ABB RobotStudio station: Sesion7_Parte1_interrupciones.rspag

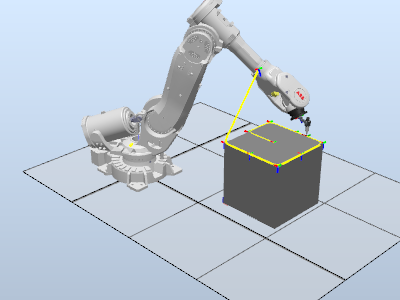
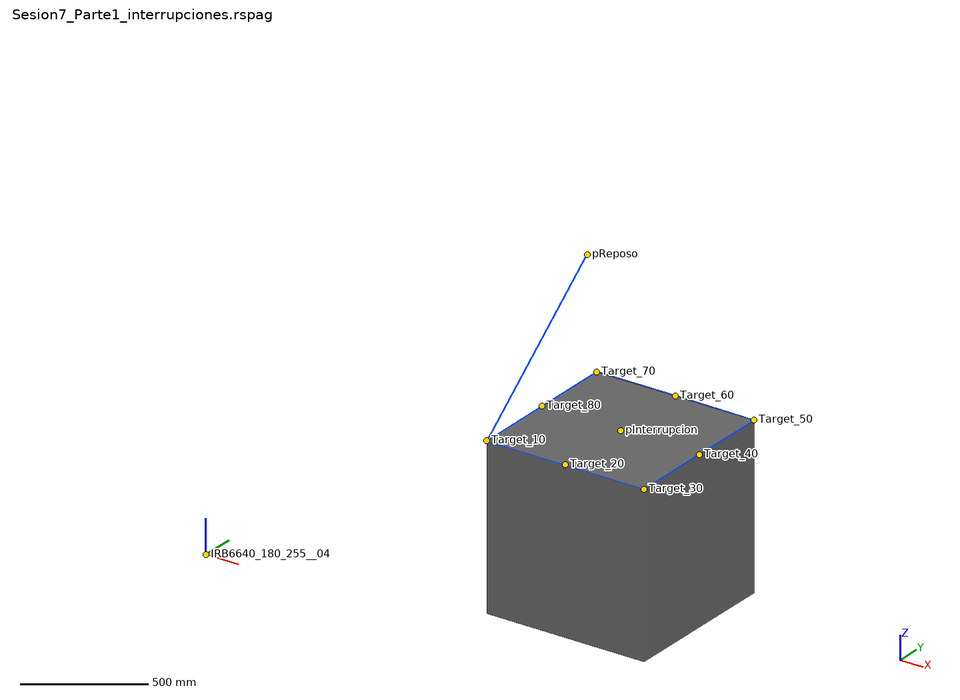
[picture v1: parts stored in the station drawn from their meshes, with robot base, taught points and paths (robot models come from the ABB library and are not in the file)]
--- station ---
Station borr (saved by RobotStudio 24.1.10713.1)
Controller Controlador10
  mechanical unit ROB_1: IRB6640_180_255__04, 6 joints, base frame (0, 0, 0) mm
Layout (positions relative to the parent item):
  - IRB6640_180_255__04 [mechanism, from %ABB.RobotStudio.Models.IRB6640%\IRB6640_180_255_G_04.rslib] at (0, 0, 0) mm; joint values [0.569, 0.4564, 0.2981, -0.9875, 0.4087, 1.4142] (rad or m)
  - MyTool [mechanism, from Training Objects\myTool.rslib] at (1608.5, 950, 950.53) mm, rotated rx -180 ry 38 rz 180 deg
  - Pieza_1 [part], size 750 x 750 x 750 mm
Attachment: MyTool is attached to IRB6640_180_255__04 / Link6
Targets, tools, work objects and paths stored in the station and not in the controller backup, written as RAPID:
! task T_ROB1
MODULE Module1
  PROC Path_10()
    MoveL pReposo,v1000,z100,MyTool\WObj:=wobj0;
    MoveL Target_10,v1000,z100,MyTool\WObj:=Workobject_1;
    MoveL Target_20,v1000,z100,MyTool\WObj:=Workobject_1;
    MoveL Target_30,v1000,z100,MyTool\WObj:=Workobject_1;
    MoveL Target_40,v1000,z100,MyTool\WObj:=Workobject_1;
    MoveL Target_50,v1000,z100,MyTool\WObj:=Workobject_1;
    MoveL Target_60,v1000,z100,MyTool\WObj:=Workobject_1;
    MoveL Target_70,v1000,z100,MyTool\WObj:=Workobject_1;
    MoveL Target_80,v1000,z100,MyTool\WObj:=Workobject_1;
    MoveL pInterrupcion,v1000,z100,MyTool\WObj:=Workobject_1;
  ENDPROC
ENDMODULE


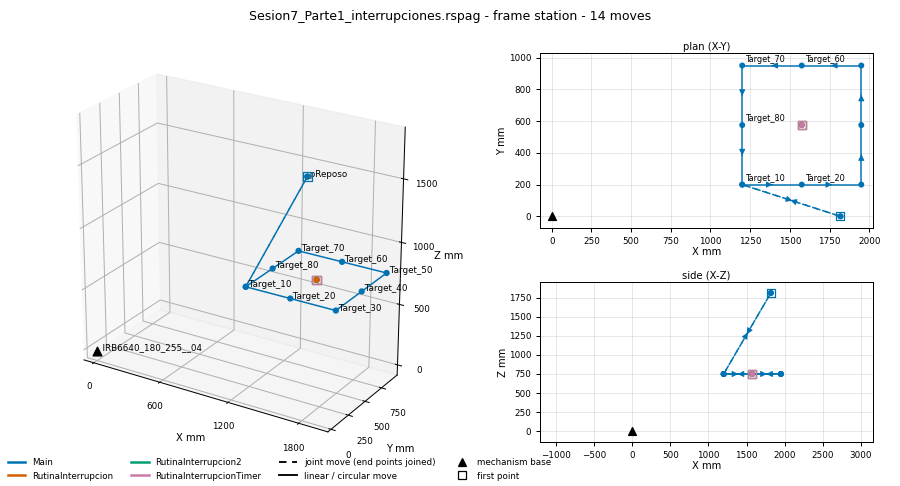
[picture p0: tool path of Sesion7_Parte1_interrupciones.rspag in frame station, 14 of 17 moves have a stored position in this frame; points joined in program order, loops and branches not executed]
--- Backups/Controlador10/RAPID/TASK1/PROGMOD/CalibData.mod ---
MODULE CalibData
    PERS tooldata MyTool:=[TRUE,[[31.792631019,0,229.638935148],[0.945518576,0,0.325568154,0]],[1,[0,0,1],[1,0,0,0],0,0,0]];
    TASK PERS wobjdata Workobject_1:=[FALSE,TRUE,"",[[1200,200,0],[1,0,0,0]],[[0,0,0],[1,0,0,0]]];
ENDMODULE

--- Backups/Controlador10/RAPID/TASK1/PROGMOD/Module1.mod ---
MODULE Module1
    CONST robtarget pReposo:=[[1818.681916784,0,1812.64730631],[0.190808996,0,0.981627183,0],[0,0,0,0],[9E+09,9E+09,9E+09,9E+09,9E+09,9E+09]];
    CONST robtarget Target_10:=[[0,0,750],[0,0,1,0],[0,-1,0,0],[9E+09,9E+09,9E+09,9E+09,9E+09,9E+09]];
    CONST robtarget Target_20:=[[375,0,750],[0,0,1,0],[0,-1,0,0],[9E+09,9E+09,9E+09,9E+09,9E+09,9E+09]];
    CONST robtarget Target_30:=[[750,0,750],[0,0,1,0],[0,-1,0,0],[9E+09,9E+09,9E+09,9E+09,9E+09,9E+09]];
    CONST robtarget Target_40:=[[750,375,750],[0,0,1,0],[0,-1,0,0],[9E+09,9E+09,9E+09,9E+09,9E+09,9E+09]];
    CONST robtarget Target_50:=[[750,750,750],[0,0,1,0],[0,-1,0,0],[9E+09,9E+09,9E+09,9E+09,9E+09,9E+09]];
    CONST robtarget Target_60:=[[375,750,750],[0,0,1,0],[0,-1,0,0],[9E+09,9E+09,9E+09,9E+09,9E+09,9E+09]];
    CONST robtarget Target_70:=[[0,750,750],[0,0,1,0],[0,0,0,0],[9E+09,9E+09,9E+09,9E+09,9E+09,9E+09]];
    CONST robtarget Target_80:=[[0,375,750],[0,0,1,0],[0,0,0,0],[9E+09,9E+09,9E+09,9E+09,9E+09,9E+09]];
    CONST robtarget pInterrupcion:=[[375,375,750],[0,0,1,0],[0,0,0,0],[9E+09,9E+09,9E+09,9E+09,9E+09,9E+09]];

    VAR intnum idInterrupcion;
    VAR intnum idInterrupcion2;
    VAR intnum idInterrupcionTimer;
    VAR robtarget stop_pos;


PROC Main()
    Reset SD_Interrupcion;

    CONNECT idInterrupcion WITH RutinaInterrupcion;
    ISignalDI ED_Sennal, 1, idInterrupcion;

    CONNECT idInterrupcion2 WITH RutinaInterrupcion2;
    ISignalDI ED_Sennal_stopmove, 1, idInterrupcion2;

    !CONNECT idInterrupcionTimer WITH RutinaInterrupcionTimer;
    !ITimer 10, idInterrupcionTimer;

    !ISleep idInterrupcionTimer;
    !IWatch idInterrupcionTimer;

    !IDisable;

    FOR i FROM 1 TO 20 DO
        MoveJ pReposo,v7000,z100,MyTool\WObj:=wobj0;
        MoveJ Target_10,v7000,z0,MyTool\WObj:=Workobject_1;
        MoveL Target_20,v100,z0,MyTool\WObj:=Workobject_1;
        MoveL Target_30,v100,z0,MyTool\WObj:=Workobject_1;
        MoveL Target_40,v100,z0,MyTool\WObj:=Workobject_1;
        MoveL Target_50,v100,z0,MyTool\WObj:=Workobject_1;
        MoveL Target_60,v100,z0,MyTool\WObj:=Workobject_1;
        MoveL Target_70,v100,z0,MyTool\WObj:=Workobject_1;
        MoveL Target_80,v100,z0,MyTool\WObj:=Workobject_1;
        MoveL Target_10,v100,z0,MyTool\WObj:=Workobject_1;
        MoveJ pReposo,v7000,z100,MyTool\WObj:=wobj0;
    ENDFOR
    !IEnable;
ENDPROC


TRAP RutinaInterrupcion
    SetDO SD_Interrupcion, 1;
    StorePath;
    stop_pos := CRobT(\Tool:=MyTool \WObj:=wobj0);
    MoveL pInterrupcion,v7000,z100,MyTool\WObj:=Workobject_1;

    MoveL stop_pos,v7000,fine,MyTool\WObj:=wobj0;
    RestoPath;
    StartMove;
    Reset SD_Interrupcion;
ENDTRAP


TRAP RutinaInterrupcion2
    SetDO SD_Interrupcion, 1;
    StopMove;
    StorePath;
    stop_pos := CRobT(\Tool:=MyTool \WObj:=wobj0);
    MoveL pInterrupcion,v7000,z100,MyTool\WObj:=Workobject_1;

    MoveL stop_pos,v7000,fine,MyTool\WObj:=wobj0;
    RestoPath;
    StartMove;
    Reset SD_Interrupcion;
ENDTRAP


TRAP RutinaInterrupcionTimer
    SetDO SD_Interrupcion, 1;
    StopMove;
    StorePath;
    stop_pos := CRobT(\Tool:=MyTool \WObj:=wobj0);
    MoveL pInterrupcion,v7000,z100,MyTool\WObj:=Workobject_1;

    MoveL stop_pos,v7000,fine,MyTool\WObj:=wobj0;
    RestoPath;
    StartMove;
    Reset SD_Interrupcion;
ENDTRAP

ENDMODULE

--- Backups/Controlador10/SYSPAR/EIO.cfg ---
EIO:CFG_1.0:6:1::
#
INDUSTRIAL_NETWORK:

      -Name "DeviceNet" -Label "DeviceNet Master/Slave Network" -Address "2"
#
DEVICENET_DEVICE:

      -Name "MiDeviceNet"
#
DEVICENET_INTERNAL_DEVICE:

      -Name "DN_Internal_Device" -VendorName "ABB Robotics"\
      -ProductName "DeviceNet Internal Slave Device"
#
EIO_SIGNAL:

      -Name "ED_Sennal" -SignalType "DI" -Device "MiDeviceNet"\
      -Label "ED_Sennal" -DeviceMap "0" -Access "All"

      -Name "ED_Sennal_StopMove" -SignalType "DI" -Device "MiDeviceNet"\
      -Label "ED_Sennal_StopMove" -DeviceMap "1" -Access "All"

      -Name "SD_Interrupcion" -SignalType "DO" -Device "MiDeviceNet"\
      -Label "SD_Interrupcion" -DeviceMap "0" -Access "All"
